VAR_GLOBAL CONSTANT
	MAXMODBUSBUFFER	: UINT := 200;
END_VAR

(* stored: Version 1.1.0.1
   GVL Param: Id {119f5a86-5b46-4a0b-afbd-569207154526}, ParameterList True *)
